LIN {X 0,Y 93.743,Z 439.819,A -85,B 0,C 180,E1 -30605.093,E2 -30605.093} C_VEL
LIN {X 0,Y 90.597,Z 452.162,A -85,B 0,C 180,E1 -30605.579,E2 -30605.579} C_VEL
LIN {X 0,Y 86.363,Z 463.788,A -85,B 0,C 180,E1 -30606.231,E2 -30606.231} C_VEL
LIN {X 0,Y 80.56,Z 475.795,A -85,B 0,C 180,E1 -30607.119,E2 -30607.119} C_VEL
LIN {X 0,Y 73.731,Z 487.016,A -85,B 0,C 180,E1 -30608.553,E2 -30608.553} C_VEL
LIN {X 0,Y 66.933,Z 496.069,A -85,B 0,C 180,E1 -30610.164,E2 -30610.164} C_VEL
LIN {X 0,Y 57.768,Z 506.201,A -85,B 0,C 180,E1 -30613.294,E2 -30613.294} C_VEL
LIN {X 0,Y 48.403,Z 514.609,A -85,B 0,C 180,E1 -30617.165,E2 -30617.165} C_VEL
LIN {X 0,Y 41.691,Z 519.964,A -85,B 0,C 180,E1 -30622.021,E2 -30622.021} C_VEL
LIN {X 0,Y 32.868,Z 526.082,A -85,B 0,C 180,E1 -30631.221,E2 -30631.221} C_VEL
LIN {X 0,Y 25.44,Z 530.916,A -85,B 0,C 180,E1 -30646.331,E2 -30646.331} C_VEL
LIN {X 0,Y 20.83,Z 534.606,A -85,B 0,C 180,E1 -30670.293,E2 -30670.293} C_VEL
LIN {X 0,Y 20.182,Z 536.499,A -85,B 0,C 180,E1 -30690.011,E2 -30690.011} C_VEL
LIN {X 0,Y 20.887,Z 537.877,A -85,B 0,C 180,E1 -30709.673,E2 -30709.673} C_VEL
LIN {X 0,Y 27.847,Z 539.414,A -85,B 0,C 180,E1 -30739.223,E2 -30739.223} C_VEL
LIN {X 0,Y 33.034,Z 539.613,A -85,B 0,C 180,E1 -30748.332,E2 -30748.332} C_VEL
LIN {X 0,Y 38.876,Z 539.422,A -85,B 0,C 180,E1 -30754.687,E2 -30754.687} C_VEL
LIN {X 0,Y 51.496,Z 537.838,A -85,B 0,C 180,E1 -30762.822,E2 -30762.822} C_VEL
LIN {X 0,Y 61.996,Z 535.452,A -85,B 0,C 180,E1 -30766.895,E2 -30766.895} C_VEL
LIN {X 0,Y 74.882,Z 531.186,A -85,B 0,C 180,E1 -30770.233,E2 -30770.233} C_VEL
LIN {X 0,Y 85.156,Z 526.613,A -85,B 0,C 180,E1 -30772.056,E2 -30772.056} C_VEL
LIN {X 0,Y 97.249,Z 519.718,A -85,B 0,C 180,E1 -30773.57,E2 -30773.57} C_VEL
LIN {X 0,Y 107.655,Z 512.277,A -85,B 0,C 180,E1 -30774.609,E2 -30774.609} C_VEL
LIN {X 0,Y 116.356,Z 504.708,A -85,B 0,C 180,E1 -30775.298,E2 -30775.298} C_VEL
LIN {X 0,Y 119.835,Z 501.253,A -85,B 0,C 180,E1 -30775.579,E2 -30775.579} C_VEL
LIN {X 0,Y 119.777,Z 501.291,A -85,B 0,C 180,E1 -30775.95,E2 -30775.95} C_VEL
LIN {X 0,Y 110.864,Z 509.54,A -85,B 0,C 180,E1 -30776.815,E2 -30776.815} C_VEL
LIN {X 0,Y 100.214,Z 517.591,A -85,B 0,C 180,E1 -30777.971,E2 -30777.971} C_VEL
LIN {X 0,Y 91.376,Z 523.005,A -85,B 0,C 180,E1 -30779.191,E2 -30779.191} C_VEL
LIN {X 0,Y 80.837,Z 528.274,A -85,B 0,C 180,E1 -30781.022,E2 -30781.022} C_VEL
LIN {X 0,Y 70.402,Z 532.331,A -85,B 0,C 180,E1 -30783.33,E2 -30783.33} C_VEL
LIN {X 0,Y 59.216,Z 535.516,A -85,B 0,C 180,E1 -30786.815,E2 -30786.815} C_VEL
LIN {X 0,Y 50.095,Z 537.261,A -85,B 0,C 180,E1 -30790.853,E2 -30790.853} C_VEL
LIN {X 0,Y 43.623,Z 538.05,A -85,B 0,C 180,E1 -30794.822,E2 -30794.822} C_VEL
LIN {X 0,Y 31.659,Z 538.362,A -85,B 0,C 180,E1 -30807.37,E2 -30807.37} C_VEL
LIN {X 0,Y 28.627,Z 538.118,A -85,B 0,C 180,E1 -30812.627,E2 -30812.627} C_VEL
LIN {X 0,Y 24.336,Z 537.668,A -85,B 0,C 180,E1 -30821.312,E2 -30821.312} C_VEL
LIN {X 0,Y 17.509,Z 536.301,A -85,B 0,C 180,E1 -30840.811,E2 -30840.811} C_VEL
LIN {X 0,Y 14.278,Z 534.66,A -85,B 0,C 180,E1 -30866.807,E2 -30866.807} C_VEL
LIN {X 0,Y 15.668,Z 532.52,A -85,B 0,C 180,E1 -30895.977,E2 -30895.977} C_VEL
LIN {X 0,Y 23.156,Z 528.499,A -85,B 0,C 180,E1 -30919.34,E2 -30919.34} C_VEL
LIN {X 0,Y 33.878,Z 522.391,A -85,B 0,C 180,E1 -30931.827,E2 -30931.827} C_VEL
LIN {X 0,Y 43.659,Z 515.733,A -85,B 0,C 180,E1 -30937.746,E2 -30937.746} C_VEL
LIN {X 0,Y 53.684,Z 507.481,A -85,B 0,C 180,E1 -30941.631,E2 -30941.631} C_VEL
LIN {X 0,Y 62.188,Z 498.996,A -85,B 0,C 180,E1 -30943.848,E2 -30943.848} C_VEL
LIN {X 0,Y 70.776,Z 488.495,A -85,B 0,C 180,E1 -30945.488,E2 -30945.488} C_VEL
LIN {X 0,Y 77.667,Z 478.1,A -85,B 0,C 180,E1 -30946.579,E2 -30946.579} C_VEL
LIN {X 0,Y 83.689,Z 466.715,A -85,B 0,C 180,E1 -30947.47,E2 -30947.47} C_VEL
LIN {X 0,Y 88.543,Z 454.514,A -85,B 0,C 180,E1 -30948.344,E2 -30948.344} C_VEL
LIN {X 0,Y 92.178,Z 441.759,A -85,B 0,C 180,E1 -30948.878,E2 -30948.878} C_VEL
LIN {X 0,Y 94.38,Z 429.609,A -85,B 0,C 180,E1 -30949.142,E2 -30949.142} C_VEL
LIN {X 0,Y 94.221,Z 427.656,A -85,B 0,C 180,E1 -30953.577,E2 -30953.577} C_VEL
LIN {X 0,Y 94.273,Z 427.797,A -85,B 0,C 180,E1 -30957.33,E2 -30957.33} C_VEL
LIN {X 0,Y 94.432,Z 429.563,A -85,B 0,C 180,E1 -30960.553,E2 -30960.553} C_VEL
LIN {X 0,Y 91.932,Z 443.283,A -85,B 0,C 180,E1 -30960.868,E2 -30960.868} C_VEL
LIN {X 0,Y 87.997,Z 456.635,A -85,B 0,C 180,E1 -30961.293,E2 -30961.293} C_VEL
LIN {X 0,Y 82.617,Z 469.362,A -85,B 0,C 180,E1 -30961.839,E2 -30961.839} C_VEL
LIN {X 0,Y 76.495,Z 480.472,A -85,B 0,C 180,E1 -30962.457,E2 -30962.457} C_VEL
LIN {X 0,Y 70.392,Z 489.493,A -85,B 0,C 180,E1 -30963.294,E2 -30963.294} C_VEL
LIN {X 0,Y 63.451,Z 498.102,A -85,B 0,C 180,E1 -30964.587,E2 -30964.587} C_VEL
LIN {X 0,Y 54.835,Z 507.018,A -85,B 0,C 180,E1 -30966.68,E2 -30966.68} C_VEL
LIN {X 0,Y 45.824,Z 514.653,A -85,B 0,C 180,E1 -30969.112,E2 -30969.112} C_VEL
LIN {X 0,Y 39.572,Z 519.312,A -85,B 0,C 180,E1 -30972.392,E2 -30972.392} C_VEL
LIN {X 0,Y 29.805,Z 525.504,A -85,B 0,C 180,E1 -30979.429,E2 -30979.429} C_VEL
LIN {X 0,Y 20.855,Z 530.403,A -85,B 0,C 180,E1 -30992.619,E2 -30992.619} C_VEL
LIN {X 0,Y 14.332,Z 534.158,A -85,B 0,C 180,E1 -31020.653,E2 -31020.653} C_VEL
LIN {X 0,Y 13.064,Z 536.08,A -85,B 0,C 180,E1 -31050.016,E2 -31050.016} C_VEL
LIN {X 0,Y 14.407,Z 537.515,A -85,B 0,C 180,E1 -31079.214,E2 -31079.214} C_VEL
LIN {X 0,Y 23.818,Z 539.108,A -85,B 0,C 180,E1 -31112.295,E2 -31112.295} C_VEL
LIN {X 0,Y 29.912,Z 539.334,A -85,B 0,C 180,E1 -31120.039,E2 -31120.039} C_VEL
LIN {X 0,Y 36.404,Z 539.188,A -85,B 0,C 180,E1 -31124.876,E2 -31124.876} C_VEL
LIN {X 0,Y 49.861,Z 537.67,A -85,B 0,C 180,E1 -31130.653,E2 -31130.653} C_VEL
LIN {X 0,Y 63.602,Z 534.596,A -85,B 0,C 180,E1 -31134.012,E2 -31134.012} C_VEL
LIN {X 0,Y 74.009,Z 531.14,A -85,B 0,C 180,E1 -31135.657,E2 -31135.657} C_VEL
LIN {X 0,Y 77.491,Z 529.741,A -85,B 0,C 180,E1 -31136.092,E2 -31136.092} C_VEL
LIN {X 0,Y 77.469,Z 529.74,A -85,B 0,C 180,E1 -31136.336,E2 -31136.336} C_VEL
LIN {X 0,Y 66.807,Z 533.489,A -85,B 0,C 180,E1 -31138.049,E2 -31138.049} C_VEL
LIN {X 0,Y 56.228,Z 536.18,A -85,B 0,C 180,E1 -31140.384,E2 -31140.384} C_VEL
LIN {X 0,Y 49.245,Z 537.43,A -85,B 0,C 180,E1 -31142.487,E2 -31142.487} C_VEL
LIN {X 0,Y 42.348,Z 538.27,A -85,B 0,C 180,E1 -31145.246,E2 -31145.246} C_VEL
LIN {X 0,Y 29.994,Z 538.678,A -85,B 0,C 180,E1 -31153.55,E2 -31153.55} C_VEL
LIN {X 0,Y 22.863,Z 538.248,A -85,B 0,C 180,E1 -31162.73,E2 -31162.73} C_VEL
LIN {X 0,Y 17.41,Z 537.448,A -85,B 0,C 180,E1 -31176.141,E2 -31176.141} C_VEL
LIN {X 0,Y 13.612,Z 536.197,A -85,B 0,C 180,E1 -31198.897,E2 -31198.897} C_VEL
LIN {X 0,Y 15.489,Z 532.628,A -85,B 0,C 180,E1 -31254.848,E2 -31254.848} C_VEL
LIN {X 0,Y 15.668,Z 532.52,A -85,B 0,C 180,E1 -31255.977,E2 -31255.977} C_VEL
LIN {X 0,Y 18.682,Z 530.683,A -85,B 0,C 180,E1 -31271.903,E2 -31271.903} C_VEL
LIN {X 0,Y 24.525,Z 527.137,A -85,B 0,C 180,E1 -31291.225,E2 -31291.225} C_VEL
LIN {X 0,Y 31.659,Z 522.84,A -85,B 0,C 180,E1 -31302.404,E2 -31302.404} C_VEL
LIN {X 0,Y 36.441,Z 519.824,A -85,B 0,C 180,E1 -31305.408,E2 -31305.408} C_VEL
LIN {X 0,Y 46.682,Z 512.576,A -85,B 0,C 180,E1 -31308.096,E2 -31308.096} C_VEL
LIN {X 0,Y 57.113,Z 503.47,A -85,B 0,C 180,E1 -31309.849,E2 -31309.849} C_VEL
LIN {X 0,Y 65.849,Z 493.986,A -85,B 0,C 180,E1 -31310.815,E2 -31310.815} C_VEL
LIN {X 0,Y 73.711,Z 483.468,A -85,B 0,C 180,E1 -31311.547,E2 -31311.547} C_VEL
LIN {X 0,Y 80.709,Z 471.738,A -85,B 0,C 180,E1 -31312.077,E2 -31312.077} C_VEL
LIN {X 0,Y 86.23,Z 459.589,A -85,B 0,C 180,E1 -31312.664,E2 -31312.664} C_VEL
LIN {X 0,Y 90.32,Z 447.411,A -85,B 0,C 180,E1 -31313.184,E2 -31313.184} C_VEL
LIN {X 0,Y 93.168,Z 434.931,A -85,B 0,C 180,E1 -31313.394,E2 -31313.394} C_VEL
LIN {X 0,Y 93.202,Z 434.634,A -85,B 0,C 180,E1 -31314.536,E2 -31314.536} C_VEL
LIN {X 0,Y 93.234,Z 434.641,A -85,B 0,C 180,E1 -31316.289,E2 -31316.289} C_VEL
LIN {X 0,Y 90.269,Z 447.712,A -85,B 0,C 180,E1 -31316.502,E2 -31316.502} C_VEL
LIN {X 0,Y 85.836,Z 460.731,A -85,B 0,C 180,E1 -31316.74,E2 -31316.74} C_VEL
LIN {X 0,Y 80.051,Z 473.084,A -85,B 0,C 180,E1 -31316.966,E2 -31316.966} C_VEL
LIN {X 0,Y 72.988,Z 484.694,A -85,B 0,C 180,E1 -31317.358,E2 -31317.358} C_VEL
LIN {X 0,Y 65.05,Z 495.134,A -85,B 0,C 180,E1 -31317.847,E2 -31317.847} C_VEL
LIN {X 0,Y 56.229,Z 504.536,A -85,B 0,C 180,E1 -31318.922,E2 -31318.922} C_VEL
LIN {X 0,Y 49.192,Z 510.815,A -85,B 0,C 180,E1 -31319.78,E2 -31319.78} C_VEL
LIN {X 0,Y 44.245,Z 514.694,A -85,B 0,C 180,E1 -31320.297,E2 -31320.297} C_VEL
LIN {X 0,Y 36.926,Z 519.787,A -85,B 0,C 180,E1 -31322.428,E2 -31322.428} C_VEL
LIN {X 0,Y 28.246,Z 524.926,A -85,B 0,C 180,E1 -31325.666,E2 -31325.666} C_VEL
LIN {X 0,Y 18.036,Z 529.89,A -85,B 0,C 180,E1 -31333.115,E2 -31333.115} C_VEL
LIN {X 0,Y 8.836,Z 533.708,A -85,B 0,C 180,E1 -31357.353,E2 -31357.353} C_VEL
LIN {X 0,Y 5.953,Z 535.662,A -85,B 0,C 180,E1 -31410.036,E2 -31410.036} C_VEL
LIN {X 0,Y 8.903,Z 537.14,A -85,B 0,C 180,E1 -31462.165,E2 -31462.165} C_VEL
LIN {X 0,Y 21.453,Z 538.801,A -85,B 0,C 180,E1 -31489.409,E2 -31489.409} C_VEL
LIN {X 0,Y 35.224,Z 538.94,A -85,B 0,C 180,E1 -31496.13,E2 -31496.13} C_VEL
LIN {X 0,Y 35.184,Z 538.916,A -85,B 0,C 180,E1 -31497.228,E2 -31497.228} C_VEL
LIN {X 0,Y 28.115,Z 538.934,A -85,B 0,C 180,E1 -31499.998,E2 -31499.998} C_VEL
LIN {X 0,Y 21.145,Z 538.563,A -85,B 0,C 180,E1 -31504.245,E2 -31504.245} C_VEL
LIN {X 0,Y 14.382,Z 537.803,A -85,B 0,C 180,E1 -31512.16,E2 -31512.16} C_VEL
LIN {X 0,Y 8.306,Z 536.598,A -85,B 0,C 180,E1 -31532.158,E2 -31532.158} C_VEL
LIN {X 0,Y 7.241,Z 534.019,A -85,B 0,C 180,E1 -31618.998,E2 -31618.998} C_VEL
LIN {X 0,Y 12.227,Z 531.981,A -85,B 0,C 180,E1 -31643.587,E2 -31643.587} C_VEL
LIN {X 0,Y 22.623,Z 527.463,A -85,B 0,C 180,E1 -31658.719,E2 -31658.719} C_VEL
LIN {X 0,Y 34.591,Z 520.999,A -85,B 0,C 180,E1 -31664.789,E2 -31664.789} C_VEL
LIN {X 0,Y 36.441,Z 519.824,A -85,B 0,C 180,E1 -31665.408,E2 -31665.408} C_VEL
LIN {X 0,Y 39.45,Z 521.513,A -85,B 0,C 180,E1 -31666.343,E2 -31666.343} C_VEL
LIN {X 0,Y 39.45,Z 600,A -85,B 0,C 180,E1 -31666.343,E2 -31666.343} C_VEL
LIN {X 0,Y 39.45,Z 600,A -85,B 0,C 180,E1 -31666.343,E2 -31666.343}

QRS_NEXT_CUT()

QRS_NEXT()
QRS_HOME()

END
